PROGRAM LeftArmManualCtrlMove
VAR
	
	point												:Points;					// 当前腕关节坐标
	target_angle										:Angles;					// 臂左右电机目标角度
	manualState											:USINT;						// 手动控制状态标志位，0
	speed												:REAL := 0.5;					// 笛卡尔坐标位移速度
	x													:REAL;						// 腕关节目标位置x
	y													:REAL;						// 腕关节目标位置y
	wrist_angle											:REAL;						// 腕电机角度
	
	//左臂举升电机
	LeftArm_Lift_Jog									:MC_Jog;
	bLeftArm_Lift_Up									:BOOL;
	bLeftArm_Lift_Down									:BOOL;
	nLeftArmLiftSpeed									:LREAL:=3;					//举升电机速度
	
	LeftArm_Right_ExtPosGen_Enable						:MC_ExtSetPointGenEnable;
	LeftArm_Right_ExtPosGen_Disable                     :MC_ExtSetPointGenDisable;
	LeftArm_Left_ExtPosGen_Enable                       :MC_ExtSetPointGenEnable;
	LeftArm_Left_ExtPosGen_Disable	                    :MC_ExtSetPointGenDisable;
	LeftArm_Wrist_ExtPosGen_Enable                      :MC_ExtSetPointGenEnable;
	LeftArm_Wrist_ExtPosGen_Disable	                    :MC_ExtSetPointGenDisable;
	
	//串口
	//fb_SerialCom		:FB_SerialCom;					
	//wrist_angle_int		:INT;
	//wrist_angle_byte	:BYTE;
	
	
END_VAR

axis_LeftArm_Left();
axis_LeftArm_Right();
axis_LeftArm_Wrist();
ExtPosGen();


// 外部位置发生器失能
LeftArm_Right_ExtPosGen_Enable.Execute 		:= FALSE;
LeftArm_Right_ExtPosGen_Disable.Execute 	:= FALSE;
LeftArm_Left_ExtPosGen_Enable.Execute 		:= FALSE;
LeftArm_Left_ExtPosGen_Disable.Execute 		:= FALSE;
LeftArm_Wrist_ExtPosGen_Enable.Execute 		:= FALSE;
LeftArm_Wrist_ExtPosGen_Disable.Execute 	:= FALSE;

IF bManualCtrl_Asm_LeftArm THEN
	// 举升电机McJog
	LeftArmLiftJog();
	
	// 运动学正解出当前腕关节点坐标
	point := LeftArmFK(axis_LeftArm_Right.NcToPlc.ActPos, axis_LeftArm_Left.NcToPlc.ActPos);
	
	// 用舵机进行程序验证的串口背景通讯
	//BackgroundSerialCtrl();
	
	IF bAutoCtrl_Part_LeftWrist THEN
		
		wrist_angle := LeftArmWristIK(axis_LeftArm_Right.NcToPlc.ActPos, axis_LeftArm_Left.NcToPlc.ActPos);		// 逆解出腕电机角度

	END_IF
	

	IF bLeftArm_Forward THEN
		x := point.x;
		y := point.y + speed;
		target_angle := LeftArmIK(x, y);
		manualState := 1;
		
	ELSIF bLeftArm_Backward THEN
	
		x := point.x;
		y := point.y - speed;
		target_angle := LeftArmIK(x, y);
		manualState := 1;
		
	ELSIF bLeftArm_Left THEN
		
		x := point.x - speed;
		y := point.y;
		target_angle := LeftArmIK(x, y);
		manualState := 1;
		
	ELSIF bLeftArm_Right THEN
		
		x := point.x + speed;
		y := point.y;
		target_angle := LeftArmIK(x, y);
		manualState := 1;
		
	ELSE
		manualState := 0;
	END_IF
	
	
	
	CASE manualState OF
		0:
			LeftArm_Right_ExtPosGen_Enable.Execute 		:= FALSE;
			LeftArm_Right_ExtPosGen_Disable.Execute 	:= TRUE;
			LeftArm_Left_ExtPosGen_Enable.Execute 		:= FALSE;
			LeftArm_Left_ExtPosGen_Disable.Execute 		:= TRUE;
			LeftArm_Wrist_ExtPosGen_Enable.Execute 		:= FALSE;
			LeftArm_Wrist_ExtPosGen_Disable.Execute 	:= TRUE;
		
		1:
			LeftArm_Right_ExtPosGen_Enable.Execute := TRUE;
			LeftArm_Left_ExtPosGen_Enable.Execute := TRUE;
			LeftArm_Wrist_ExtPosGen_Enable.Execute := TRUE;
			IF axis_LeftArm_Right.Status.ExtSetPointGenEnabled AND axis_LeftArm_Left.Status.ExtSetPointGenEnabled AND axis_LeftArm_Wrist.Status.ExtSetPointGenEnabled THEN
				MC_ExtSetPointGenFeed(
					Position:= target_angle.theta1_right, 
					Velocity:= 1,  
					Acceleration:= 3,  
					Direction:= 1, 
					Axis:= axis_LeftArm_Right);
		
				MC_ExtSetPointGenFeed(
					Position:= target_angle.theta2_left, 
					Velocity:= 1,  
					Acceleration:= 3,  
					Direction:= 1, 
					Axis:= axis_LeftArm_Left);
					
				MC_ExtSetPointGenFeed(
					Position:= wrist_angle, 
					Velocity:= 1, 
					Acceleration:= 3, 
					Direction:= 1, 
					Axis:= axis_LeftArm_Wrist);
			END_IF
	END_CASE

//ELSE

END_IF

ACTION ExtPosGen:
LeftArm_Right_ExtPosGen_Enable(
	Axis:= axis_LeftArm_Right, 
	Execute:= LeftArm_Right_ExtPosGen_Enable.Execute, 
	Position:= , 
	PositionType:= , 
	Done=> , 
	Busy=> , 
	Error=> , 
	ErrorID=> , 
	Enabled=> );
	
LeftArm_Right_ExtPosGen_Disable(
	Axis:= axis_LeftArm_Right, 
	Execute:= LeftArm_Right_ExtPosGen_Disable.Execute, 
	Done=> , 
	Busy=> , 
	Error=> , 
	ErrorID=> , 
	Enabled=> );
	
LeftArm_Left_ExtPosGen_Enable(
	Axis:= axis_LeftArm_Left, 
	Execute:= LeftArm_Left_ExtPosGen_Enable.Execute, 
	Position:= , 
	PositionType:= , 
	Done=> , 
	Busy=> , 
	Error=> , 
	ErrorID=> , 
	Enabled=> );
	
LeftArm_Left_ExtPosGen_Disable(
	Axis:= axis_LeftArm_Left, 
	Execute:= LeftArm_Left_ExtPosGen_Disable.Execute, 
	Done=> , 
	Busy=> , 
	Error=> , 
	ErrorID=> , 
	Enabled=> );
	
LeftArm_Wrist_ExtPosGen_Enable(
	Axis:= axis_LeftArm_Wrist, 
	Execute:= LeftArm_Wrist_ExtPosGen_Enable.Execute, 
	Position:= , 
	PositionType:= , 
	Done=> , 
	Busy=> , 
	Error=> , 
	ErrorID=> , 
	Enabled=> );
	
LeftArm_Wrist_ExtPosGen_Disable(
	Axis:= axis_LeftArm_Wrist, 
	Execute:= LeftArm_Wrist_ExtPosGen_Disable.Execute, 
	Done=> , 
	Busy=> , 
	Error=> , 
	ErrorID=> , 
	Enabled=> );
END_ACTION

ACTION LeftArmLiftJog:
LeftArm_Lift_Jog(
	Axis:= axis_LeftArm_Lift, 
	JogForward:= bLeftArm_Lift_Up, 
	JogBackwards:= bLeftArm_Lift_Down, 
	Mode:= MC_JOGMODE_CONTINOUS, 
	Position:= , 
	Velocity:= nLeftArmLiftSpeed, 
	Acceleration:= , 
	Deceleration:= , 
	Jerk:= , 
	Done=> , 
	Busy=> , 
	Active=> , 
	CommandAborted=> , 
	Error=> , 
	ErrorID=> );
END_ACTION

END_PROGRAM

(* stored: Version 1.1.0.1, ProductVersion 3.1.4024.14
   POU LeftArmManualCtrlMove: Id {7ce4e0af-3646-41d7-be69-9b2292beb16d}, SpecialFunc None
   Action ExtPosGen: Id {e3c908b9-5d30-4d3c-9346-9279cf2bd814}
   Action LeftArmLiftJog: Id {fa2827fa-9b6c-474c-aa67-a14473c70902} *)
